(* IEC 61131-3 sources: Lasal/CPU_5344_V01/Class/GlobalListGreat, 1 file *)

(* ---- GlobalListGreat.st ---- *)
(*!
<Class
	Name               = "GlobalListGreat"
	Revision           = "0.0"
	RealtimeTask       = "false"
	CyclicTask         = "false"
	BackgroundTask     = "false"
	Sigmatek           = "false"
	OSInterface        = "false"
	HighPriority       = "false"
	Automatic          = "false"
	UpdateMode         = "Prescan"
	SharedCommandTable = "true"
	Objectsize         = "(284,120)">
	<Channels>
		<Server Name="ClassSvr" Visualized="false" Initialize="false" WriteProtected="true" Retentive="false"/>
		<Server Name="ClassSvr0" Class="GlobalList" Visualized="false" Initialize="false" WriteProtected="true" Retentive="false"/>
		<Client Name="ListAanvoer" Required="true" Internal="true"/>
		<Client Name="RamSregels1" Required="true" Internal="true"/>
		<Client Name="RamSregels10" Required="true" Internal="true"/>
		<Client Name="RamSregels11" Required="true" Internal="true"/>
		<Client Name="RamSregels12" Required="true" Internal="true"/>
		<Client Name="RamSregels13" Required="true" Internal="true"/>
		<Client Name="RamSregels14" Required="true" Internal="true"/>
		<Client Name="RamSregels15" Required="true" Internal="true"/>
		<Client Name="RamSregels16" Required="true" Internal="true"/>
		<Client Name="RamSregels17" Required="true" Internal="true"/>
		<Client Name="RamSregels18" Required="true" Internal="true"/>
		<Client Name="RamSregels19" Required="true" Internal="true"/>
		<Client Name="RamSregels2" Required="true" Internal="true"/>
		<Client Name="RamSregels20" Required="true" Internal="true"/>
		<Client Name="RamSregels21" Required="true" Internal="true"/>
		<Client Name="RamSregels22" Required="true" Internal="true"/>
		<Client Name="RamSregels23" Required="true" Internal="true"/>
		<Client Name="RamSregels24" Required="true" Internal="true"/>
		<Client Name="RamSregels25" Required="true" Internal="true"/>
		<Client Name="RamSregels26" Required="true" Internal="true"/>
		<Client Name="RamSregels27" Required="true" Internal="true"/>
		<Client Name="RamSregels28" Required="true" Internal="true"/>
		<Client Name="RamSregels29" Required="true" Internal="true"/>
		<Client Name="RamSregels3" Required="true" Internal="true"/>
		<Client Name="RamSregels30" Required="true" Internal="true"/>
		<Client Name="RamSregels31" Required="true" Internal="true"/>
		<Client Name="RamSregels32" Required="true" Internal="true"/>
		<Client Name="RamSregels4" Required="true" Internal="true"/>
		<Client Name="RamSregels5" Required="true" Internal="true"/>
		<Client Name="RamSregels6" Required="true" Internal="true"/>
		<Client Name="RamSregels7" Required="true" Internal="true"/>
		<Client Name="RamSregels8" Required="true" Internal="true"/>
		<Client Name="RamSregels9" Required="true" Internal="true"/>
	</Channels>
	<Network Name="GlobalListGreat">
		<!-- List of Components in this network -->
		<Components>
			<Object
				Name           = "ListAanvoer"
				Class          = "GlobalList"
				Position       = "(1650,120)"
				Visualized     = "false"
				BackgroundTime = "10 ms">
				<Channels>
					<Server Name="ActRegel"/>
					<Server Name="ClassSvr"/>
					<Server Name="FileRegel"/>
					<Server Name="Stepper"/>
					<Client Name="Aanv" Value="1"/>
					<Client Name="FileSys"/>
					<Client Name="ram1"/>
					<Client Name="ram10"/>
					<Client Name="ram2"/>
					<Client Name="ram3"/>
					<Client Name="ram4"/>
					<Client Name="ram5"/>
					<Client Name="ram6"/>
					<Client Name="ram7"/>
					<Client Name="ram8"/>
					<Client Name="ram9"/>
				</Channels>
			</Object>
			<Object
				Name       = "RamSregels1"
				Class      = "RamSregels"
				Position   = "(300,90)"
				Visualized = "false">
				<Channels>
					<Server Name="ClassSvr"/>
				</Channels>
			</Object>
			<Object
				Name       = "RamSregels10"
				Class      = "RamSregels"
				Position   = "(300,1170)"
				Visualized = "false">
				<Channels>
					<Server Name="ClassSvr"/>
				</Channels>
			</Object>
			<Object
				Name       = "RamSregels11"
				Class      = "RamSregels"
				Position   = "(300,1290)"
				Visualized = "false">
				<Channels>
					<Server Name="ClassSvr"/>
				</Channels>
			</Object>
			<Object
				Name       = "RamSregels12"
				Class      = "RamSregels"
				Position   = "(300,1410)"
				Visualized = "false">
				<Channels>
					<Server Name="ClassSvr"/>
				</Channels>
			</Object>
			<Object
				Name       = "RamSregels13"
				Class      = "RamSregels"
				Position   = "(300,1530)"
				Visualized = "false">
				<Channels>
					<Server Name="ClassSvr"/>
				</Channels>
			</Object>
			<Object
				Name       = "RamSregels14"
				Class      = "RamSregels"
				Position   = "(300,1650)"
				Visualized = "false">
				<Channels>
					<Server Name="ClassSvr"/>
				</Channels>
			</Object>
			<Object
				Name       = "RamSregels15"
				Class      = "RamSregels"
				Position   = "(300,1770)"
				Visualized = "false">
				<Channels>
					<Server Name="ClassSvr"/>
				</Channels>
			</Object>
			<Object
				Name       = "RamSregels16"
				Class      = "RamSregels"
				Position   = "(300,1890)"
				Visualized = "false">
				<Channels>
					<Server Name="ClassSvr"/>
				</Channels>
			</Object>
			<Object
				Name       = "RamSregels17"
				Class      = "RamSregels"
				Position   = "(300,2010)"
				Visualized = "false">
				<Channels>
					<Server Name="ClassSvr"/>
				</Channels>
			</Object>
			<Object
				Name       = "RamSregels18"
				Class      = "RamSregels"
				Position   = "(300,2130)"
				Visualized = "false">
				<Channels>
					<Server Name="ClassSvr"/>
				</Channels>
			</Object>
			<Object
				Name       = "RamSregels19"
				Class      = "RamSregels"
				Position   = "(300,2250)"
				Visualized = "false">
				<Channels>
					<Server Name="ClassSvr"/>
				</Channels>
			</Object>
			<Object
				Name       = "RamSregels2"
				Class      = "RamSregels"
				Position   = "(300,210)"
				Visualized = "false">
				<Channels>
					<Server Name="ClassSvr"/>
				</Channels>
			</Object>
			<Object
				Name       = "RamSregels20"
				Class      = "RamSregels"
				Position   = "(300,2370)"
				Visualized = "false">
				<Channels>
					<Server Name="ClassSvr"/>
				</Channels>
			</Object>
			<Object
				Name       = "RamSregels21"
				Class      = "RamSregels"
				Position   = "(300,2490)"
				Visualized = "false">
				<Channels>
					<Server Name="ClassSvr"/>
				</Channels>
			</Object>
			<Object
				Name       = "RamSregels22"
				Class      = "RamSregels"
				Position   = "(300,2610)"
				Visualized = "false">
				<Channels>
					<Server Name="ClassSvr"/>
				</Channels>
			</Object>
			<Object
				Name       = "RamSregels23"
				Class      = "RamSregels"
				Position   = "(300,2730)"
				Visualized = "false">
				<Channels>
					<Server Name="ClassSvr"/>
				</Channels>
			</Object>
			<Object
				Name       = "RamSregels24"
				Class      = "RamSregels"
				Position   = "(300,2850)"
				Visualized = "false">
				<Channels>
					<Server Name="ClassSvr"/>
				</Channels>
			</Object>
			<Object
				Name       = "RamSregels25"
				Class      = "RamSregels"
				Position   = "(300,2970)"
				Visualized = "false">
				<Channels>
					<Server Name="ClassSvr"/>
				</Channels>
			</Object>
			<Object
				Name       = "RamSregels26"
				Class      = "RamSregels"
				Position   = "(300,3090)"
				Visualized = "false">
				<Channels>
					<Server Name="ClassSvr"/>
				</Channels>
			</Object>
			<Object
				Name       = "RamSregels27"
				Class      = "RamSregels"
				Position   = "(300,3210)"
				Visualized = "false">
				<Channels>
					<Server Name="ClassSvr"/>
				</Channels>
			</Object>
			<Object
				Name       = "RamSregels28"
				Class      = "RamSregels"
				Position   = "(300,3330)"
				Visualized = "false">
				<Channels>
					<Server Name="ClassSvr"/>
				</Channels>
			</Object>
			<Object
				Name       = "RamSregels29"
				Class      = "RamSregels"
				Position   = "(300,3450)"
				Visualized = "false">
				<Channels>
					<Server Name="ClassSvr"/>
				</Channels>
			</Object>
			<Object
				Name       = "RamSregels3"
				Class      = "RamSregels"
				Position   = "(300,330)"
				Visualized = "false">
				<Channels>
					<Server Name="ClassSvr"/>
				</Channels>
			</Object>
			<Object
				Name       = "RamSregels30"
				Class      = "RamSregels"
				Position   = "(300,3570)"
				Visualized = "false">
				<Channels>
					<Server Name="ClassSvr"/>
				</Channels>
			</Object>
			<Object
				Name       = "RamSregels31"
				Class      = "RamSregels"
				Position   = "(300,3690)"
				Visualized = "false">
				<Channels>
					<Server Name="ClassSvr"/>
				</Channels>
			</Object>
			<Object
				Name       = "RamSregels32"
				Class      = "RamSregels"
				Position   = "(300,3810)"
				Visualized = "false">
				<Channels>
					<Server Name="ClassSvr"/>
				</Channels>
			</Object>
			<Object
				Name       = "RamSregels4"
				Class      = "RamSregels"
				Position   = "(300,450)"
				Visualized = "false">
				<Channels>
					<Server Name="ClassSvr"/>
				</Channels>
			</Object>
			<Object
				Name       = "RamSregels5"
				Class      = "RamSregels"
				Position   = "(300,570)"
				Visualized = "false">
				<Channels>
					<Server Name="ClassSvr"/>
				</Channels>
			</Object>
			<Object
				Name       = "RamSregels6"
				Class      = "RamSregels"
				Position   = "(300,690)"
				Visualized = "false">
				<Channels>
					<Server Name="ClassSvr"/>
				</Channels>
			</Object>
			<Object
				Name       = "RamSregels7"
				Class      = "RamSregels"
				Position   = "(300,810)"
				Visualized = "false">
				<Channels>
					<Server Name="ClassSvr"/>
				</Channels>
			</Object>
			<Object
				Name       = "RamSregels8"
				Class      = "RamSregels"
				Position   = "(300,930)"
				Visualized = "false">
				<Channels>
					<Server Name="ClassSvr"/>
				</Channels>
			</Object>
			<Object
				Name       = "RamSregels9"
				Class      = "RamSregels"
				Position   = "(300,1050)"
				Visualized = "false">
				<Channels>
					<Server Name="ClassSvr"/>
				</Channels>
			</Object>
		</Components>
		<Comments>
		</Comments>
		<!-- List of Connections in this network -->
		<Connections>
			<Connection Source="this.ListAanvoer" Destination="ListAanvoer.ClassSvr"/>
			<Connection Source="this.RamSregels5" Destination="RamSregels5.ClassSvr"/>
			<Connection Source="this.RamSregels4" Destination="RamSregels4.ClassSvr"/>
			<Connection Source="this.RamSregels2" Destination="RamSregels2.ClassSvr"/>
			<Connection Source="this.RamSregels1" Destination="RamSregels1.ClassSvr"/>
			<Connection Source="this.RamSregels3" Destination="RamSregels3.ClassSvr"/>
			<Connection Source="this.ClassSvr0" Destination="ListAanvoer.ClassSvr" Vertices="(2122,270),(1950,210),"/>
			<Connection Source="ListAanvoer.ram1" Destination="RamSregels1.ClassSvr" Vertices="(1650,330),(690,330),(690,180),(600,180),"/>
			<Connection Source="ListAanvoer.ram2" Destination="RamSregels2.ClassSvr" Vertices="(1650,390),(660,390),(660,300),(600,300),"/>
			<Connection Source="ListAanvoer.ram3" Destination="RamSregels3.ClassSvr" Vertices="(1650,450),(630,450),(630,420),(600,420),"/>
			<Connection Source="ListAanvoer.ram4" Destination="RamSregels4.ClassSvr" Vertices="(1650,510),(630,510),(630,540),(600,540),"/>
			<Connection Source="ListAanvoer.ram5" Destination="RamSregels5.ClassSvr" Vertices="(1650,570),(660,570),(660,660),(600,660),"/>
			<Connection Source="this.RamSregels6" Destination="RamSregels6.ClassSvr"/>
			<Connection Source="this.RamSregels7" Destination="RamSregels7.ClassSvr"/>
			<Connection Source="this.RamSregels8" Destination="RamSregels8.ClassSvr"/>
			<Connection Source="this.RamSregels9" Destination="RamSregels9.ClassSvr"/>
			<Connection Source="this.RamSregels10" Destination="RamSregels10.ClassSvr"/>
			<Connection Source="ListAanvoer.ram6" Destination="RamSregels6.ClassSvr" Vertices="(1650,630),(690,630),(690,780),(600,780),"/>
			<Connection Source="ListAanvoer.ram7" Destination="RamSregels7.ClassSvr" Vertices="(1650,690),(720,690),(720,900),(600,900),"/>
			<Connection Source="ListAanvoer.ram8" Destination="RamSregels8.ClassSvr" Vertices="(1650,750),(750,750),(750,1020),(600,1020),"/>
			<Connection Source="ListAanvoer.ram9" Destination="RamSregels9.ClassSvr" Vertices="(1650,810),(780,810),(780,1140),(570,1140),(600,1140),"/>
			<Connection Source="ListAanvoer.ram10" Destination="RamSregels10.ClassSvr" Vertices="(1650,870),(810,870),(810,1260),(600,1260),"/>
			<Connection Source="this.RamSregels11" Destination="RamSregels11.ClassSvr"/>
			<Connection Source="this.RamSregels13" Destination="RamSregels13.ClassSvr"/>
			<Connection Source="this.RamSregels16" Destination="RamSregels16.ClassSvr"/>
			<Connection Source="this.RamSregels15" Destination="RamSregels15.ClassSvr"/>
			<Connection Source="this.RamSregels17" Destination="RamSregels17.ClassSvr"/>
			<Connection Source="this.RamSregels14" Destination="RamSregels14.ClassSvr"/>
			<Connection Source="this.RamSregels12" Destination="RamSregels12.ClassSvr"/>
			<Connection Source="this.RamSregels18" Destination="RamSregels18.ClassSvr"/>
			<Connection Source="this.RamSregels19" Destination="RamSregels19.ClassSvr"/>
			<Connection Source="this.RamSregels21" Destination="RamSregels21.ClassSvr"/>
			<Connection Source="this.RamSregels24" Destination="RamSregels24.ClassSvr"/>
			<Connection Source="this.RamSregels20" Destination="RamSregels20.ClassSvr"/>
			<Connection Source="this.RamSregels22" Destination="RamSregels22.ClassSvr"/>
			<Connection Source="this.RamSregels23" Destination="RamSregels23.ClassSvr"/>
			<Connection Source="this.RamSregels25" Destination="RamSregels25.ClassSvr"/>
			<Connection Source="this.RamSregels26" Destination="RamSregels26.ClassSvr"/>
			<Connection Source="this.RamSregels27" Destination="RamSregels27.ClassSvr"/>
			<Connection Source="this.RamSregels31" Destination="RamSregels31.ClassSvr"/>
			<Connection Source="this.RamSregels28" Destination="RamSregels28.ClassSvr"/>
			<Connection Source="this.RamSregels29" Destination="RamSregels29.ClassSvr"/>
			<Connection Source="this.RamSregels30" Destination="RamSregels30.ClassSvr"/>
			<Connection Source="this.RamSregels32" Destination="RamSregels32.ClassSvr"/>
		</Connections>
		<!-- Headerfiles -->
		<Options>
		</Options>
	</Network>
</Class>
*)
GlobalListGreat : CLASS
  //Servers:
	ClassSvr 	: SvrChCmd_DINT;
	ClassSvr0 	: SvrChCmd_DINT;
  //Clients:
	ListAanvoer 	: CltChCmd_GlobalList;
	RamSregels2 	: CltChCmd_RamSregels;
	RamSregels1 	: CltChCmd_RamSregels;
	RamSregels3 	: CltChCmd_RamSregels;
	RamSregels4 	: CltChCmd_RamSregels;
	RamSregels5 	: CltChCmd_RamSregels;
	RamSregels6 	: CltChCmd_RamSregels;
	RamSregels7 	: CltChCmd_RamSregels;
	RamSregels8 	: CltChCmd_RamSregels;
	RamSregels9 	: CltChCmd_RamSregels;
	RamSregels10 	: CltChCmd_RamSregels;
	RamSregels11 	: CltChCmd_RamSregels;
	RamSregels12 	: CltChCmd_RamSregels;
	RamSregels13 	: CltChCmd_RamSregels;
	RamSregels14 	: CltChCmd_RamSregels;
	RamSregels15 	: CltChCmd_RamSregels;
	RamSregels16 	: CltChCmd_RamSregels;
	RamSregels17 	: CltChCmd_RamSregels;
	RamSregels18 	: CltChCmd_RamSregels;
	RamSregels19 	: CltChCmd_RamSregels;
	RamSregels20 	: CltChCmd_RamSregels;
	RamSregels21 	: CltChCmd_RamSregels;
	RamSregels22 	: CltChCmd_RamSregels;
	RamSregels23 	: CltChCmd_RamSregels;
	RamSregels24 	: CltChCmd_RamSregels;
	RamSregels25 	: CltChCmd_RamSregels;
	RamSregels26 	: CltChCmd_RamSregels;
	RamSregels27 	: CltChCmd_RamSregels;
	RamSregels28 	: CltChCmd_RamSregels;
	RamSregels29 	: CltChCmd_RamSregels;
	RamSregels30 	: CltChCmd_RamSregels;
	RamSregels31 	: CltChCmd_RamSregels;
	RamSregels32 	: CltChCmd_RamSregels;
  //Variables:
  //Functions:

	FUNCTION VIRTUAL GLOBAL ClassSvr0::Read
		VAR_OUTPUT
			output (EAX) 	: DINT;
		END_VAR;
  //Tables:
	FUNCTION @STD
		VAR_OUTPUT
			ret_code	: CONFSTATES;
		END_VAR;
	FUNCTION GLOBAL TAB @CT_;
END_CLASS;

#pragma using GlobalList
#pragma using RamSregels

FUNCTION VIRTUAL GLOBAL GlobalListGreat::ClassSvr0::Read
	VAR_OUTPUT
		output (EAX) 	: DINT;
	END_VAR

	ClassSvr0 := ListAanvoer.ClassSvr.Read();
	output := ClassSvr0;

END_FUNCTION
